// TIA Portal V19 export
FUNCTION "A0303_Spintore_CALL" : Void   // FC144, LAD
// stored: SetENOAutomatically false
BEGIN

REGION Network 1: <<< LATO TESTA >>>
END_REGION

REGION Network 2: Data In - Spintore Verticale
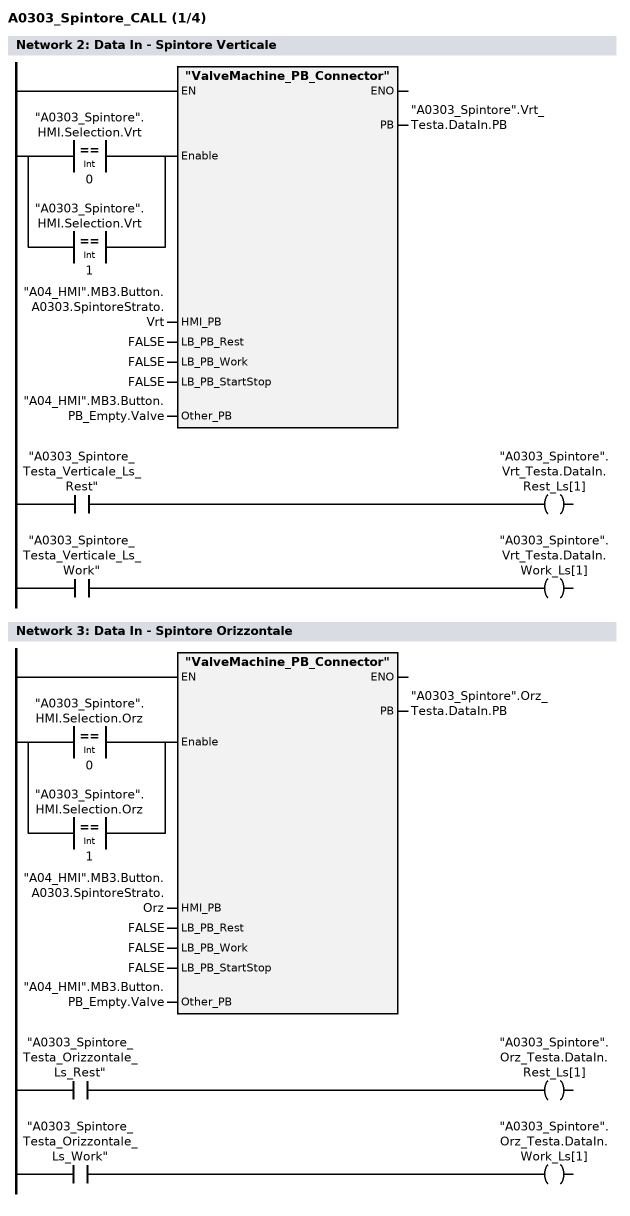
   RUNG wire#powerrail
      "ValveMachine_PB_Connector"(Enable := wire#w1, HMI_PB := "A04_HMI".MB3.Button.A0303.SpintoreStrato.Vrt, LB_PB_Rest := FALSE, LB_PB_Work := FALSE, LB_PB_StartStop := FALSE, Other_PB := "A04_HMI".MB3.Button.PB_Empty.Valve, PB => "A0303_Spintore".Vrt_Testa.DataIn.PB)
   END_RUNG
   RUNG wire#powerrail
      { S7_Templates := "SrcType := Int" } EQ_Contact(in1 := "A0303_Spintore".HMI.Selection.Vrt, in2 := 0)
   END_RUNG wire#w1
   RUNG wire#powerrail
      { S7_Templates := "SrcType := Int" } EQ_Contact(in1 := "A0303_Spintore".HMI.Selection.Vrt, in2 := 1)
   END_RUNG wire#w1
   RUNG wire#powerrail
      Contact( "A0303_Spintore_Testa_Verticale_Ls_Rest" )
      Coil( "A0303_Spintore".Vrt_Testa.DataIn.Rest_Ls[1] )
   END_RUNG
   RUNG wire#powerrail
      Contact( "A0303_Spintore_Testa_Verticale_Ls_Work" )
      Coil( "A0303_Spintore".Vrt_Testa.DataIn.Work_Ls[1] )
   END_RUNG
   // the same network as SCL:
   "ValveMachine_PB_Connector"(Enable := ("A0303_Spintore".HMI.Selection.Vrt = 0) OR ("A0303_Spintore".HMI.Selection.Vrt = 1),
                           HMI_PB := "A04_HMI".MB3.Button.A0303.SpintoreStrato.Vrt,
                           LB_PB_Rest := FALSE,
                           LB_PB_Work := FALSE,
                           LB_PB_StartStop := FALSE,
                           Other_PB := "A04_HMI".MB3.Button.PB_Empty.Valve,
                           PB => "A0303_Spintore".Vrt_Testa.DataIn.PB);
   "A0303_Spintore".Vrt_Testa.DataIn.Rest_Ls[1] := "A0303_Spintore_Testa_Verticale_Ls_Rest";
   "A0303_Spintore".Vrt_Testa.DataIn.Work_Ls[1] := "A0303_Spintore_Testa_Verticale_Ls_Work";
END_REGION

REGION Network 3: Data In - Spintore Orizzontale
   RUNG wire#powerrail
      "ValveMachine_PB_Connector"(Enable := wire#w1, HMI_PB := "A04_HMI".MB3.Button.A0303.SpintoreStrato.Orz, LB_PB_Rest := FALSE, LB_PB_Work := FALSE, LB_PB_StartStop := FALSE, Other_PB := "A04_HMI".MB3.Button.PB_Empty.Valve, PB => "A0303_Spintore".Orz_Testa.DataIn.PB)
   END_RUNG
   RUNG wire#powerrail
      { S7_Templates := "SrcType := Int" } EQ_Contact(in1 := "A0303_Spintore".HMI.Selection.Orz, in2 := 0)
   END_RUNG wire#w1
   RUNG wire#powerrail
      { S7_Templates := "SrcType := Int" } EQ_Contact(in1 := "A0303_Spintore".HMI.Selection.Orz, in2 := 1)
   END_RUNG wire#w1
   RUNG wire#powerrail
      Contact( "A0303_Spintore_Testa_Orizzontale_Ls_Rest" )
      Coil( "A0303_Spintore".Orz_Testa.DataIn.Rest_Ls[1] )
   END_RUNG
   RUNG wire#powerrail
      Contact( "A0303_Spintore_Testa_Orizzontale_Ls_Work" )
      Coil( "A0303_Spintore".Orz_Testa.DataIn.Work_Ls[1] )
   END_RUNG
   // the same network as SCL:
   "ValveMachine_PB_Connector"(Enable := ("A0303_Spintore".HMI.Selection.Orz = 0) OR ("A0303_Spintore".HMI.Selection.Orz = 1),
                           HMI_PB := "A04_HMI".MB3.Button.A0303.SpintoreStrato.Orz,
                           LB_PB_Rest := FALSE,
                           LB_PB_Work := FALSE,
                           LB_PB_StartStop := FALSE,
                           Other_PB := "A04_HMI".MB3.Button.PB_Empty.Valve,
                           PB => "A0303_Spintore".Orz_Testa.DataIn.PB);
   "A0303_Spintore".Orz_Testa.DataIn.Rest_Ls[1] := "A0303_Spintore_Testa_Orizzontale_Ls_Rest";
   "A0303_Spintore".Orz_Testa.DataIn.Work_Ls[1] := "A0303_Spintore_Testa_Orizzontale_Ls_Work";
END_REGION

REGION Network 4: <<< LATO CODA >>>
END_REGION

REGION Network 5: Data In - Spintore Verticale
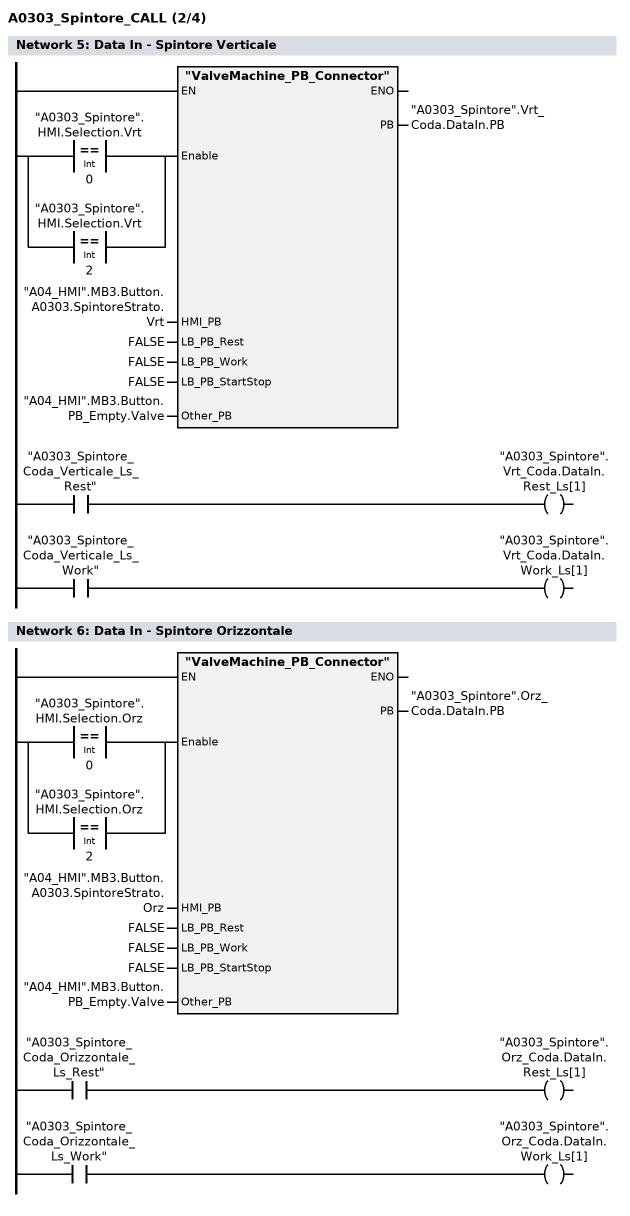
   RUNG wire#powerrail
      "ValveMachine_PB_Connector"(Enable := wire#w1, HMI_PB := "A04_HMI".MB3.Button.A0303.SpintoreStrato.Vrt, LB_PB_Rest := FALSE, LB_PB_Work := FALSE, LB_PB_StartStop := FALSE, Other_PB := "A04_HMI".MB3.Button.PB_Empty.Valve, PB => "A0303_Spintore".Vrt_Coda.DataIn.PB)
   END_RUNG
   RUNG wire#powerrail
      { S7_Templates := "SrcType := Int" } EQ_Contact(in1 := "A0303_Spintore".HMI.Selection.Vrt, in2 := 0)
   END_RUNG wire#w1
   RUNG wire#powerrail
      { S7_Templates := "SrcType := Int" } EQ_Contact(in1 := "A0303_Spintore".HMI.Selection.Vrt, in2 := 2)
   END_RUNG wire#w1
   RUNG wire#powerrail
      Contact( "A0303_Spintore_Coda_Verticale_Ls_Rest" )
      Coil( "A0303_Spintore".Vrt_Coda.DataIn.Rest_Ls[1] )
   END_RUNG
   RUNG wire#powerrail
      Contact( "A0303_Spintore_Coda_Verticale_Ls_Work" )
      Coil( "A0303_Spintore".Vrt_Coda.DataIn.Work_Ls[1] )
   END_RUNG
   // the same network as SCL:
   "ValveMachine_PB_Connector"(Enable := ("A0303_Spintore".HMI.Selection.Vrt = 0) OR ("A0303_Spintore".HMI.Selection.Vrt = 2),
                           HMI_PB := "A04_HMI".MB3.Button.A0303.SpintoreStrato.Vrt,
                           LB_PB_Rest := FALSE,
                           LB_PB_Work := FALSE,
                           LB_PB_StartStop := FALSE,
                           Other_PB := "A04_HMI".MB3.Button.PB_Empty.Valve,
                           PB => "A0303_Spintore".Vrt_Coda.DataIn.PB);
   "A0303_Spintore".Vrt_Coda.DataIn.Rest_Ls[1] := "A0303_Spintore_Coda_Verticale_Ls_Rest";
   "A0303_Spintore".Vrt_Coda.DataIn.Work_Ls[1] := "A0303_Spintore_Coda_Verticale_Ls_Work";
END_REGION

REGION Network 6: Data In - Spintore Orizzontale
   RUNG wire#powerrail
      "ValveMachine_PB_Connector"(Enable := wire#w1, HMI_PB := "A04_HMI".MB3.Button.A0303.SpintoreStrato.Orz, LB_PB_Rest := FALSE, LB_PB_Work := FALSE, LB_PB_StartStop := FALSE, Other_PB := "A04_HMI".MB3.Button.PB_Empty.Valve, PB => "A0303_Spintore".Orz_Coda.DataIn.PB)
   END_RUNG
   RUNG wire#powerrail
      { S7_Templates := "SrcType := Int" } EQ_Contact(in1 := "A0303_Spintore".HMI.Selection.Orz, in2 := 0)
   END_RUNG wire#w1
   RUNG wire#powerrail
      { S7_Templates := "SrcType := Int" } EQ_Contact(in1 := "A0303_Spintore".HMI.Selection.Orz, in2 := 2)
   END_RUNG wire#w1
   RUNG wire#powerrail
      Contact( "A0303_Spintore_Coda_Orizzontale_Ls_Rest" )
      Coil( "A0303_Spintore".Orz_Coda.DataIn.Rest_Ls[1] )
   END_RUNG
   RUNG wire#powerrail
      Contact( "A0303_Spintore_Coda_Orizzontale_Ls_Work" )
      Coil( "A0303_Spintore".Orz_Coda.DataIn.Work_Ls[1] )
   END_RUNG
   // the same network as SCL:
   "ValveMachine_PB_Connector"(Enable := ("A0303_Spintore".HMI.Selection.Orz = 0) OR ("A0303_Spintore".HMI.Selection.Orz = 2),
                           HMI_PB := "A04_HMI".MB3.Button.A0303.SpintoreStrato.Orz,
                           LB_PB_Rest := FALSE,
                           LB_PB_Work := FALSE,
                           LB_PB_StartStop := FALSE,
                           Other_PB := "A04_HMI".MB3.Button.PB_Empty.Valve,
                           PB => "A0303_Spintore".Orz_Coda.DataIn.PB);
   "A0303_Spintore".Orz_Coda.DataIn.Rest_Ls[1] := "A0303_Spintore_Coda_Orizzontale_Ls_Rest";
   "A0303_Spintore".Orz_Coda.DataIn.Work_Ls[1] := "A0303_Spintore_Coda_Orizzontale_Ls_Work";
END_REGION

REGION Network 8: Data In - OP
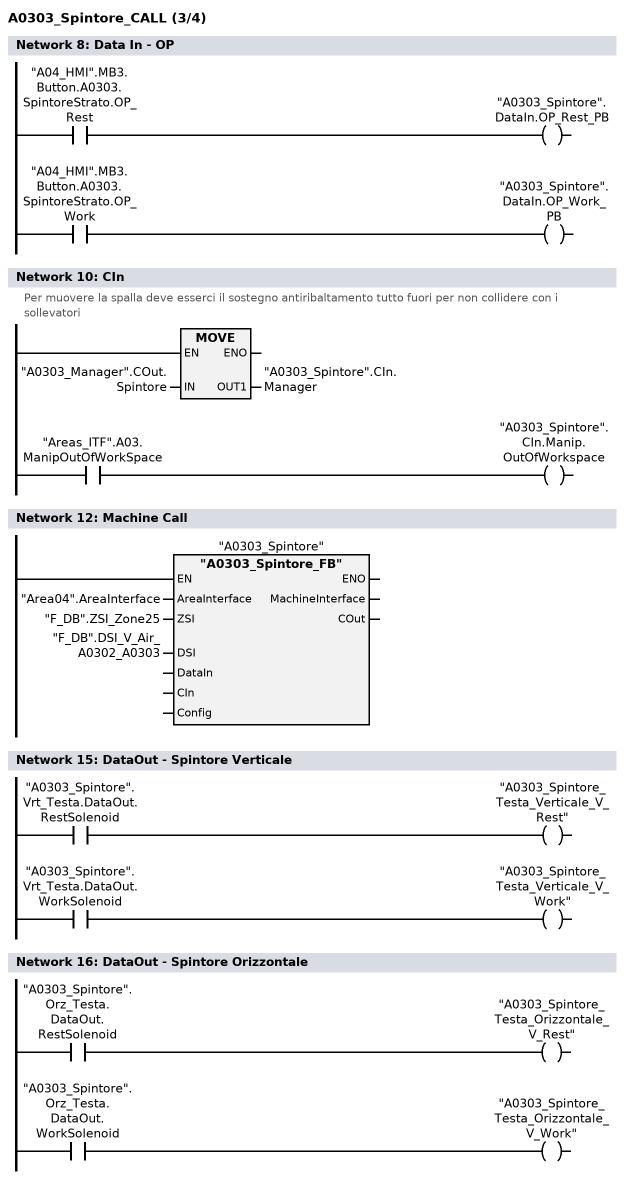
   RUNG wire#powerrail
      Contact( "A04_HMI".MB3.Button.A0303.SpintoreStrato.OP_Rest )
      Coil( "A0303_Spintore".DataIn.OP_Rest_PB )
   END_RUNG
   RUNG wire#powerrail
      Contact( "A04_HMI".MB3.Button.A0303.SpintoreStrato.OP_Work )
      Coil( "A0303_Spintore".DataIn.OP_Work_PB )
   END_RUNG
   // the same network as SCL:
   "A0303_Spintore".DataIn.OP_Rest_PB := "A04_HMI".MB3.Button.A0303.SpintoreStrato.OP_Rest;
   "A0303_Spintore".DataIn.OP_Work_PB := "A04_HMI".MB3.Button.A0303.SpintoreStrato.OP_Work;
END_REGION

REGION Network 10: CIn
   // Per muovere la spalla deve esserci il sostegno antiribaltamento tutto fuori per non collidere con i sollevatori
   RUNG wire#powerrail
      Move(in := "A0303_Manager".COut.Spintore, out1 => "A0303_Spintore".CIn.Manager)
   END_RUNG
   RUNG wire#powerrail
      Contact( "Areas_ITF".A03.ManipOutOfWorkSpace )
      Coil( "A0303_Spintore".CIn.Manip.OutOfWorkspace )
   END_RUNG
   // the same network as SCL:
   "A0303_Spintore".CIn.Manager := "A0303_Manager".COut.Spintore;
   "A0303_Spintore".CIn.Manip.OutOfWorkspace := "Areas_ITF".A03.ManipOutOfWorkSpace;
END_REGION

REGION Network 11: >
END_REGION

REGION Network 12: Machine Call
   RUNG wire#powerrail
      "A0303_Spintore"(AreaInterface := "Area04".AreaInterface, ZSI := "F_DB".ZSI_Zone25, DSI := "F_DB".DSI_V_Air_A0302_A0303, DataIn :=, CIn :=, MachineInterface =>, COut =>, Config :=)
   END_RUNG
   // the same network as SCL:
   "A0303_Spintore"(AreaInterface := "Area04".AreaInterface,   // "A0303_Spintore_FB"
                    ZSI := "F_DB".ZSI_Zone25,
                    DSI := "F_DB".DSI_V_Air_A0302_A0303);
END_REGION

REGION Network 14: <<< LATO TESTA >>>
END_REGION

REGION Network 15: DataOut - Spintore Verticale
   RUNG wire#powerrail
      Contact( "A0303_Spintore".Vrt_Testa.DataOut.RestSolenoid )
      Coil( "A0303_Spintore_Testa_Verticale_V_Rest" )
   END_RUNG
   RUNG wire#powerrail
      Contact( "A0303_Spintore".Vrt_Testa.DataOut.WorkSolenoid )
      Coil( "A0303_Spintore_Testa_Verticale_V_Work" )
   END_RUNG
   // the same network as SCL:
   "A0303_Spintore_Testa_Verticale_V_Rest" := "A0303_Spintore".Vrt_Testa.DataOut.RestSolenoid;
   "A0303_Spintore_Testa_Verticale_V_Work" := "A0303_Spintore".Vrt_Testa.DataOut.WorkSolenoid;
END_REGION

REGION Network 16: DataOut - Spintore Orizzontale
   RUNG wire#powerrail
      Contact( "A0303_Spintore".Orz_Testa.DataOut.RestSolenoid )
      Coil( "A0303_Spintore_Testa_Orizzontale_V_Rest" )
   END_RUNG
   RUNG wire#powerrail
      Contact( "A0303_Spintore".Orz_Testa.DataOut.WorkSolenoid )
      Coil( "A0303_Spintore_Testa_Orizzontale_V_Work" )
   END_RUNG
   // the same network as SCL:
   "A0303_Spintore_Testa_Orizzontale_V_Rest" := "A0303_Spintore".Orz_Testa.DataOut.RestSolenoid;
   "A0303_Spintore_Testa_Orizzontale_V_Work" := "A0303_Spintore".Orz_Testa.DataOut.WorkSolenoid;
END_REGION

REGION Network 17: <<< LATO CODA >>>
END_REGION

REGION Network 18: DataOut - Spintore Verticale
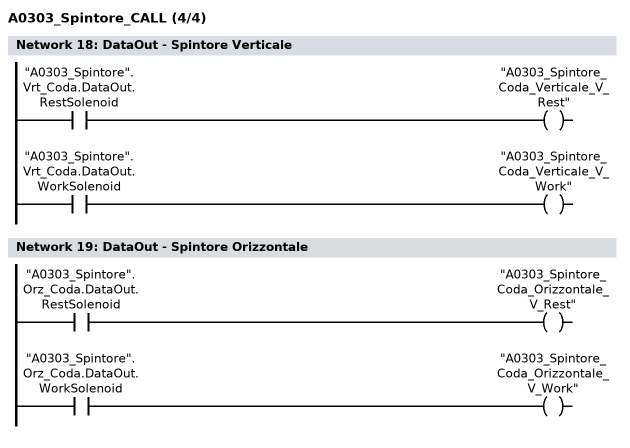
   RUNG wire#powerrail
      Contact( "A0303_Spintore".Vrt_Coda.DataOut.RestSolenoid )
      Coil( "A0303_Spintore_Coda_Verticale_V_Rest" )
   END_RUNG
   RUNG wire#powerrail
      Contact( "A0303_Spintore".Vrt_Coda.DataOut.WorkSolenoid )
      Coil( "A0303_Spintore_Coda_Verticale_V_Work" )
   END_RUNG
   // the same network as SCL:
   "A0303_Spintore_Coda_Verticale_V_Rest" := "A0303_Spintore".Vrt_Coda.DataOut.RestSolenoid;
   "A0303_Spintore_Coda_Verticale_V_Work" := "A0303_Spintore".Vrt_Coda.DataOut.WorkSolenoid;
END_REGION

REGION Network 19: DataOut - Spintore Orizzontale
   RUNG wire#powerrail
      Contact( "A0303_Spintore".Orz_Coda.DataOut.RestSolenoid )
      Coil( "A0303_Spintore_Coda_Orizzontale_V_Rest" )
   END_RUNG
   RUNG wire#powerrail
      Contact( "A0303_Spintore".Orz_Coda.DataOut.WorkSolenoid )
      Coil( "A0303_Spintore_Coda_Orizzontale_V_Work" )
   END_RUNG
   // the same network as SCL:
   "A0303_Spintore_Coda_Orizzontale_V_Rest" := "A0303_Spintore".Orz_Coda.DataOut.RestSolenoid;
   "A0303_Spintore_Coda_Orizzontale_V_Work" := "A0303_Spintore".Orz_Coda.DataOut.WorkSolenoid;
END_REGION
END_FUNCTION
